Fanuc KAREL source: kx00033.KL

-- PROVISIONAL review KL for V940-1; original PC SHA256 eb9a6348389e80500b5d3e4a76979499ec518df4d06f569927ed735f33edf256
-- Incomplete behavior may be omitted. Consult companion uncertainty JSON. Do not deploy.
PROGRAM KX00033
%NOLOCKGROUP
-- UNRESOLVED_DECL I type=fa0010
-- UNRESOLVED_DECL J type=fa0010
-- UNRESOLVED_DECL B type=fa0012
-- UNRESOLVED_DECL F type=fa001d
-- UNRESOLVED_DECL S type=fa1f50
-- UNRESOLVED_DECL P type=fa0102
BEGIN
  -- V9_ZERO_TABLE_METADATA_HINT layout=0001; no indexed target words; source/name/runtime held
  -- UNRESOLVED_PC offsets 5-12; opcodes 9D,23
  -- UNRESOLVED_PC offsets 17-21; opcodes 7F
END KX00033
